FUNCTION_BLOCK ABSTRACT FB_SensorDecoratorTestParent EXTENDS FB_BaseComponentDecoratorParent IMPLEMENTS ITF_SensorDecoratorTest
VAR
	bContactTest			: BOOL;
END_VAR

(*			
	EVERDE sp. z o.o.
	Rafał Osajda		05.02.2025		TC 4026.13		wer. 0.0.0.1
	Zwraca aktualny stan czujnika
*)
METHOD IsActive : BOOL
END_METHOD

METHOD SetContract
VAR_INPUT
	bIN: BOOL;
END_VAR
THIS^.bContactTest		:= bIN;
END_METHOD

END_FUNCTION_BLOCK

(* stored: Version 1.1.0.1
   POU FB_SensorDecoratorTestParent: Id {67645e76-427e-4501-bf87-8b0f905c7add}, SpecialFunc None
   Method IsActive: Id {d21918fa-2e53-0edb-3f50-08a193727751}
   Method SetContract: Id {2400656c-d1fa-4d75-9e59-2914639345c5} *)
